// TIA Portal V19 export
FUNCTION_BLOCK "TYPIC_C103_IF_OVN"   // FB16, FBD
TITLE = TYPIC_C103_IF_OVN: LSB NB
{ S7_Optimized_Access := 'TRUE' }
AUTHOR : OCOTECH
FAMILY : Typical
NAME : C103.704
// Logisch Object Besturing: C103.805
// 
// De interne functie laagspanningsverdeelbord no break in dienstkoker verzorgt de bewaking van een laagspanningsverdeelbord no break in dienstkoker.
// stored: MemoryReserve 10, SetENOAutomatically false
   VAR_INPUT
      EXT_AUT { ExternalAccessible := 'False'; ExternalVisible := 'False'; ExternalWritable := 'False'} : Bool;   // Externe (hoofd) beveiliging (1 = OK)
      EXT_HW { ExternalAccessible := 'False'; ExternalVisible := 'False'; ExternalWritable := 'False'} : Bool;   // Sturings hardware (PLC) bewaking (1 = OK)
      IN_SCL1 { ExternalAccessible := 'False'; ExternalVisible := 'False'; ExternalWritable := 'False'} : Bool;   // Standmelding aankomstschakelaar normaal
      IN_SCL2 { ExternalAccessible := 'False'; ExternalVisible := 'False'; ExternalWritable := 'False'} : Bool;   // Standmelding aankomstschakelaar no-break
      IN_BEV { ExternalAccessible := 'False'; ExternalVisible := 'False'; ExternalWritable := 'False'} : Bool;   // Standmelding automaat kast verwarming en ventilatie
   END_VAR
   VAR_OUTPUT
      VAR_IF_OVN { ExternalAccessible := 'False'; ExternalVisible := 'False'; ExternalWritable := 'False'} : "C103_VAR_IF_OVN_TYPIC";   // Struct met alle variabelen naar bovenliggende functies
   END_VAR
   VAR
      STO { ExternalWritable := 'False'} : Struct   // Storingen
         A001 { ExternalAccessible := 'False'; ExternalVisible := 'False'} : Bool;   // Laagspanningsverdeelbord no break in dienstkoker beveiliging aangesproken
         A002 { ExternalAccessible := 'False'; ExternalVisible := 'False'} : Bool;   // Laagspanningsverdeelbord no break in dienstkoker in storing
      END_STRUCT;
      VAR { ExternalWritable := 'False'} : Struct   // Variabelen
         SCL1 { ExternalAccessible := 'False'; ExternalVisible := 'False'} : Bool;   // Standmelding aankomstschakelaar normaal
         SCL2 { ExternalAccessible := 'False'; ExternalVisible := 'False'} : Bool;   // Standmelding aankomstschakelaar no-break
         BEV { ExternalAccessible := 'False'; ExternalVisible := 'False'} : Bool;   // Standmelding automaat kast verwarming en ventilatie
      END_STRUCT;
   END_VAR
BEGIN

REGION Network 1: START
END_REGION

REGION Network 2: +++ Verwerking meetwaarden en statussen +++
   // De meetwaarde en status wordt ontvangen vanuit de interne sturing.
END_REGION

REGION Network 3: +++ Storingen +++
   // Combinatie van de storingen
END_REGION

REGION Network 4: Storing A001: Laagspanningsverdeelbord no break in dienstkoker beveiliging aangesproken
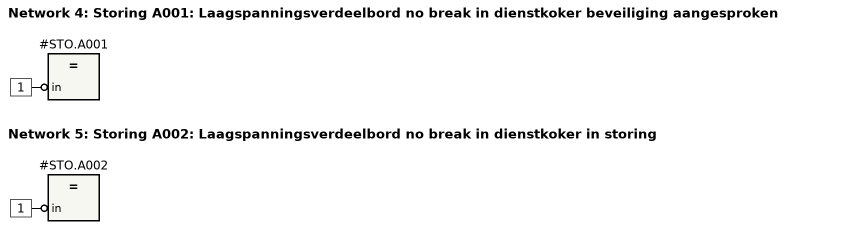
   #STO.A001 := NOT 1;
END_REGION

REGION Network 5: Storing A002: Laagspanningsverdeelbord no break in dienstkoker in storing
   #STO.A002 := NOT 1;
END_REGION

REGION Network 6 (SCL): EINDE
   // Variabelen van intern scada rakvlak naar outputs copieren
   #VAR_IF_OVN.SCL1 := #VAR.SCL1;
   #VAR_IF_OVN.SCL2 := #VAR.SCL2;
   #VAR_IF_OVN.BEV := #VAR.BEV;
END_REGION
END_FUNCTION_BLOCK
